(* CoDeSys 2.3 export: FTURNONK16PUMP.EXP *)

(* POU K16/fTurnOnK16Pump, ST *)
FUNCTION fTurnOnK16Pump : BOOL
VAR_INPUT
	PumpID : USINT;
END_VAR
fSetK16Pump(TRUE, PumpID);
END_FUNCTION
